TYPE THeaterState :
STRUCT
	EnableOut : BOOL;
	HeatingOut : REAL;
	AutCtrl : BOOL;
	ManCtrl : BOOL;
	Err 	: BOOL;
	StateInt : INT;
	GenErr : BOOL; //signalisation: error occured

	HeatingPower : REAL;
	

END_STRUCT
END_TYPE

(* stored: Version 1.1.0.1, ProductVersion 3.1.4024.12
   DUT THeaterState: Id {d83d7e51-3b95-4d8a-aaac-7196e3c7e3d2} *)
